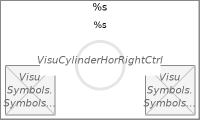
VISUALIZATION VisuCylinderTurn  // 200x120
VAR_IN_OUT
	fbVisuCylinder: FB_VISU_CYLINDER;
END_VAR
    Textfield (0,15 200x20), "%s", text variable: fbVisuCylinder.strInfo, colour toggle: fbVisuCylinder.stEvent.bEventActive
    Textfield (0,0 200x14), "%s", text variable: fbVisuCylinder.strFullObjName
    Image (145,65 50x50), invisible if: fbVisuCylinder.bWorkArrowInvisible, image: VisuSymbols.Symbols.ArrowHalfRightDown
        p2175578022: fbVisuCylinder.dwFrameColorWork
    Image (5,65 50x50), invisible if: fbVisuCylinder.bBaseArrowInvisible, image: VisuSymbols.Symbols.ArrowHalfLeftRight
        p2175578022: fbVisuCylinder.dwFrameColorBase
    RoundedRectangle (40,55 120x20)
        p2858320360: fbVisuCylinder.iAngle
    Ellipse (75,40 50x50)
        OnMouseClick: execute { fbVisuCylinder.bFrameInvisible:=false; }
    Frame (0,0 200x120), invisible if: fbVisuCylinder.bFrameInvisible, frame switch variable: fbVisuCylinder.iFrame
        shows VisuCylinderHorRightCtrl(fbVisuCylinder := fbVisuCylinder)
END_VISUALIZATION

(* stored: Version 1.1.0.1, ProductVersion 3.1.4024.12
   Visu VisuCylinderTurn: Id {0c2f1c73-0774-4373-ad83-b9db7839169b} *)
